(* CODESYS project Projekt_Wytwornia_Soku_Jerzy_Batygolski.project

Project tree, tasks and I/O mapping:
  Device : Berghof MX6 Control, Berghof Automation GmbH, version 1.21.0.0
    application Application
      libraries: Standard, 3.5.9.0 (System); Util, 3.5.11.0 (System); VisuUserMgmtDialogs, 3.5.10.0 (System); VisuDialogs, * (System); CAA Memory Block Manager Extern, 3.5.13.0 (CAA Technical Workgroup)
      task Control_program (cyclic, interval t#25ms, priority 1) calls CTRL_PRG
      task Simulation_program (cyclic, interval t#25ms, priority 1) calls SIM_PRG
      task VISU_TASK (cyclic, interval 50 ms, priority 31) calls VisuElems.Visu_Prg
      task TrendRecordingTask (cyclic, interval 100 ms, priority 31) calls VisuTrendStorageAccess.GlobalInstances.g_TrendRecordingManager.CyclicCall
      task AlarmManagerTask (cyclic, interval 50 ms, priority 31) calls AlarmManager.Alarm_Prg
      program SIM_PRG [ST]
      ENUMS/
        data type ConveyorStateEnum
        data type FillerStateEnum
        data type PasteurizationTankStateEnum
        data type PressStateEnum
        data type InnerFillerStateEnum
      MACHINE_STRUCTS/
        data type ConveyorMachineType
        data type PressMachineType
        data type PasteurizationTankType
        data type FillerMachineType
      STRUCTS/
        Conveyor/
          data type ConveyorCmdType
          data type ConveyorFailureType
          data type ConveyorSensorType
          data type ConveyorFlagType
          data type ConveyorParamType
        Press/
          data type PressCmdType
          data type PressFailureType
          data type PressSensorType
          data type PressFlagType
          data type PressParamType
        PasteurizationTank/
          data type PasteurCmdType
          data type PasteurFailureType
          data type PasteurSensorType
          data type PasteurFlagType
        Filler/
          data type FillerCmdType
          data type FillerFailureType
          data type FillerSensorType
          data type FillerFlagType
        Apple/
          data type AppleType
        Failure/
          data type FailureType
      image pool ImagePool
      program CTRL_PRG [ST]
      visualisation MainPage
      global variables GlobalVar
      visualisation Trends
      visualisation Alarms
      visualisation ErrorService
      Alarm Configuration
        alarm class ConvError (priority 10, acknowledge REP_ACK)
        alarm class TankLevelHigh (priority 30, acknowledge REP)
        AlarmStorage
        text list Conv
        alarm group Conv
            0 [ConvError]: Comparison Equal, ExpressionToCompare TRUE, Expression GlobalVar.Conveyor.Failure.ConvError.Active - "Conveyor is stuck"
            1 [GrinderError]: Comparison Equal, ExpressionToCompare TRUE, Expression GlobalVar.Conveyor.Failure.GrinderError.Active - "Grinder is stuck"
            2 [ConvEStop]: Comparison Equal, ExpressionToCompare TRUE, Expression GlobalVar.Conveyor.Failure.EStopPressed.Active - "Conveyor emergency stop is pressed"
            3 [GroundBuffer]: Comparison Equal, ExpressionToCompare TRUE, Expression GlobalVar.Conveyor.Failure.GroundBufferLevelTooHigh.Active - "Ground buffer level (<LATCH1> kg) is too high"
        alarm class GrinderError (priority 10, acknowledge REP_ACK)
        alarm class ConvEStop (priority 10, acknowledge REP_ACK)
        alarm class GroundBuffer (priority 10, acknowledge REP_ACK)
        alarm class PressError (priority 10, acknowledge REP_ACK)
        text list Press
        alarm group Press
            0 [PressError]: Comparison Equal, ExpressionToCompare TRUE, Expression GlobalVar.Press.Failure.PressError.Active - "Press is stucked"
            1 [TankBuffer]: Comparison Equal, ExpressionToCompare TRUE, Expression GlobalVar.Press.Failure.BufferTankLevelTooHigh.Active - "Buffer tank level (<LATCH1> l) is too high"
            2 [PressEStop]: Comparison Equal, ExpressionToCompare TRUE, Expression GlobalVar.Press.Failure.EStopPressed.Active - "Press emergency stop is pressed"
            3 [TankLevelHigh]: Comparison Equal, ExpressionToCompare TRUE, Expression GlobalVar.Press.Flag.TankLevelHigh - "Buffer tank level (<LATCH1> l) is high"
        text list PasteurizationTank
        alarm group PasteurizationTank
            0 [HeatingError]: Comparison Equal, ExpressionToCompare TRUE, Expression GlobalVar.PasteurTank.Failure.HeatingError.Active - "Heater is damaged"
            1 [PasteurEStop]: Comparison Equal, ExpressionToCompare TRUE, Expression GlobalVar.PasteurTank.Failure.EStopPressed.Active - "Pasteurization emergency stop is pressed"
        text list FillingMachine
        alarm group FillingMachine
            0 [CapError]: Comparison Equal, ExpressionToCompare TRUE, Expression GlobalVar.Filler.Failure.CapError.Active - "Cap is stuck"
            1 [FillError]: Comparison Equal, ExpressionToCompare TRUE, Expression GlobalVar.Filler.Failure.FillError.Active - "Filler is stuck"
            2 [FillerEStop]: Comparison Equal, ExpressionToCompare TRUE, Expression GlobalVar.Filler.Failure.EStopPressed.Active - "Filler emergency stop is pressed"
        alarm class TankBuffer (priority 10, acknowledge REP_ACK)
        alarm class PressEStop (priority 10, acknowledge REP_ACK)
        alarm class HeatingError (priority 10, acknowledge REP_ACK)
        alarm class PasteurEStop (priority 10, acknowledge REP_ACK)
        alarm class CapError (priority 10, acknowledge REP_ACK)
        alarm class FillError (priority 10, acknowledge REP_ACK)
        alarm class FillerEStop (priority 10, acknowledge REP_ACK)
  libraries: VisuSymbols, 3.5.10.0 (System)
  text list GlobalTextList
  5ce3da45-db07-42e7-a21c-a00fff4ed8f6|C:\Users\Jurek\Desktop\logo.png
  5ce3da45-db07-42e7-a21c-a00fff4ed8f6|C:\Users\Jurek\Desktop\Estop.png
  5ce3da45-db07-42e7-a21c-a00fff4ed8f6|C:\Users\Jurek\Desktop\Grafiki\EstopBtn2.jpg
  5ce3da45-db07-42e7-a21c-a00fff4ed8f6|C:\Users\Jurek\Desktop\Grafiki\EstopBtn2Pressed.jpg
  5ce3da45-db07-42e7-a21c-a00fff4ed8f6|C:\Users\Jurek\Desktop\Grafiki\Myjka_MT_1000.jpg
  5ce3da45-db07-42e7-a21c-a00fff4ed8f6|C:\Users\Jurek\Desktop\Grafiki\jablkaLevel3.png
  5ce3da45-db07-42e7-a21c-a00fff4ed8f6|C:\Users\Jurek\Desktop\Grafiki\jablkaLevel2.png
  5ce3da45-db07-42e7-a21c-a00fff4ed8f6|C:\Users\Jurek\Desktop\Grafiki\jablkaLevel1.png
  5ce3da45-db07-42e7-a21c-a00fff4ed8f6|C:\Users\Jurek\Desktop\Grafiki\jablkaLevel4.png
  5ce3da45-db07-42e7-a21c-a00fff4ed8f6|C:\Users\Jurek\Desktop\Grafiki\jablko5full.png
  5ce3da45-db07-42e7-a21c-a00fff4ed8f6|C:\Users\Jurek\Desktop\Grafiki\jablka_zmielone.png
  5ce3da45-db07-42e7-a21c-a00fff4ed8f6|C:\Users\Jurek\Desktop\Grafiki\prasaPNGgotowa.png
  5ce3da45-db07-42e7-a21c-a00fff4ed8f6|C:\Users\Jurek\Desktop\Grafiki\prasa\maleKolo.png
  5ce3da45-db07-42e7-a21c-a00fff4ed8f6|C:\Users\Jurek\Desktop\Grafiki\prasa\duzeKolo.png
  5ce3da45-db07-42e7-a21c-a00fff4ed8f6|C:\Users\Jurek\Desktop\Grafiki\prasa\nDuzeKolo.png
  5ce3da45-db07-42e7-a21c-a00fff4ed8f6|C:\Users\Jurek\Desktop\Grafiki\prasa\nMaleKolo.png
  5ce3da45-db07-42e7-a21c-a00fff4ed8f6|C:\Users\Jurek\Desktop\Grafiki\prasa\sok.png
  5ce3da45-db07-42e7-a21c-a00fff4ed8f6|C:\Users\Jurek\Desktop\Grafiki\prasa\zbiornik1500L.png
  5ce3da45-db07-42e7-a21c-a00fff4ed8f6|C:\Users\Jurek\Desktop\Grafiki\prasa\tank1000L.png
  5ce3da45-db07-42e7-a21c-a00fff4ed8f6|C:\Users\Jurek\Desktop\Grafiki\prasa\tank1002L.png
  5ce3da45-db07-42e7-a21c-a00fff4ed8f6|C:\Users\Jurek\Desktop\Grafiki\header.png
  5ce3da45-db07-42e7-a21c-a00fff4ed8f6|C:\Users\Jurek\Desktop\Grafiki\AlarmIcon.png
  5ce3da45-db07-42e7-a21c-a00fff4ed8f6|C:\Users\Jurek\Desktop\Grafiki\AlarmIcon2.png
*)

// Device/Application/ENUMS/ConveyorStateEnum
{attribute 'qualified_only'}
{attribute 'strict'}
TYPE ConveyorStateEnum :
(
	STATE_IDLE,
	STATE_WORKING,
	STATE_ERROR
);
END_TYPE

// Device/Application/ENUMS/FillerStateEnum
{attribute 'qualified_only'}
{attribute 'strict'}
TYPE FillerStateEnum :
(
	STATE_IDLE,
	STATE_WORKING,
	STATE_ERROR
);
END_TYPE

// Device/Application/ENUMS/PasteurizationTankStateEnum
{attribute 'qualified_only'}
{attribute 'strict'}
TYPE PasteurizationTankStateEnum :
(
	STATE_IDLE,
	STATE_FILLING,
	STATE_PASTEUR,
	STATE_ERROR
);
END_TYPE

// Device/Application/ENUMS/PressStateEnum
{attribute 'qualified_only'}
{attribute 'strict'}
TYPE PressStateEnum :
(
	STATE_IDLE,
	STATE_WORKING,
	STATE_ERROR
);
END_TYPE

// Device/Application/MACHINE_STRUCTS/ConveyorMachineType
TYPE ConveyorMachineType :
STRUCT
	Cmd: ConveyorCmdType;
	Failure: ConveyorFailureType;
	Sensor: ConveyorSensorType;
	State: ConveyorStateEnum;
	Flag: ConveyorFlagType;
	Param: ConveyorParamType;
END_STRUCT
END_TYPE

// Device/Application/MACHINE_STRUCTS/PressMachineType
TYPE PressMachineType :
STRUCT
	Cmd: PressCmdType;
	Failure: PressFailureType;
	Sensor: PressSensorType;
	State: PressStateEnum;
	Flag: PressFlagType;
	Param: PressParamType;
END_STRUCT
END_TYPE

// Device/Application/MACHINE_STRUCTS/PasteurizationTankType
TYPE PasteurizationTankType :
STRUCT
	Cmd: PasteurCmdType;
	Failure: PasteurFailureType;
	Sensor: PasteurSensorType;
	State: PasteurizationTankStateEnum;
	Flag: PasteurFlagType;
END_STRUCT
END_TYPE

// Device/Application/MACHINE_STRUCTS/FillerMachineType
TYPE FillerMachineType :
STRUCT
	Cmd: FillerCmdType;
	Failure: FillerFailureType;
	Sensor: FillerSensorType;
	State: FillerStateEnum;
	SimState: InnerFillerStateEnum;
	Flag: FillerFlagType;
END_STRUCT
END_TYPE

// Device/Application/STRUCTS/Conveyor/ConveyorCmdType
TYPE ConveyorCmdType :
STRUCT
	Start: BOOL;
	Stop: BOOL;
	EStop: BOOL;
	RunConv: BOOL;
END_STRUCT
END_TYPE

// Device/Application/STRUCTS/Conveyor/ConveyorFailureType
TYPE ConveyorFailureType :
STRUCT
	ConvError: FailureType;
	GrinderError: FailureType;
	EStopPressed: FailureType;
	GroundBufferLevelTooHigh: FailureType;
END_STRUCT
END_TYPE

// Device/Application/STRUCTS/Conveyor/ConveyorSensorType
TYPE ConveyorSensorType :
STRUCT
	Weight: REAL;
	GrinderRunning: BOOL;
END_STRUCT
END_TYPE

// Device/Application/STRUCTS/Conveyor/ConveyorFlagType
TYPE ConveyorFlagType :
STRUCT
	ProcessError: BOOL;
	ApplesOnConveyor: BOOL;
END_STRUCT
END_TYPE

// Device/Application/STRUCTS/Press/PressCmdType
TYPE PressCmdType :
STRUCT
	Start: BOOL;
	Stop: BOOL;
	EStop: BOOL;
	PressRun: BOOL;
END_STRUCT
END_TYPE

// Device/Application/STRUCTS/Press/PressFailureType
TYPE PressFailureType :
STRUCT
	PressError: FailureType;
	BufferTankLevelTooHigh: FailureType;
	EStopPressed: FailureType;
END_STRUCT
END_TYPE

// Device/Application/STRUCTS/Press/PressSensorType
TYPE PressSensorType :
STRUCT
	GroundBufferLevel: REAL;
	TotalJuiceProduced: REAL;
	TankLevel: REAL;
END_STRUCT
END_TYPE

// Device/Application/STRUCTS/Press/PressFlagType
TYPE PressFlagType :
STRUCT
	ProcessError: BOOL;
	TankLevelHigh: BOOL;
END_STRUCT
END_TYPE

// Device/Application/STRUCTS/PasteurizationTank/PasteurCmdType
TYPE PasteurCmdType :
STRUCT
	Start: BOOL;
	Stop: BOOL;
	EStop: BOOL;
	Fill: BOOL;
	Heat: BOOL;
	Cool: BOOL;
END_STRUCT
END_TYPE

// Device/Application/STRUCTS/PasteurizationTank/PasteurFailureType
TYPE PasteurFailureType :
STRUCT
	HeatingError: FailureType;
	EStopPressed: FailureType;
END_STRUCT
END_TYPE

// Device/Application/STRUCTS/PasteurizationTank/PasteurSensorType
TYPE PasteurSensorType :
STRUCT
	TankLevel: REAL;
	TargetTemp: REAL;
	ActTemp: LREAL;
END_STRUCT
END_TYPE

// Device/Application/STRUCTS/PasteurizationTank/PasteurFlagType
TYPE PasteurFlagType :
STRUCT
	ProcessError: BOOL;
	Filling: BOOL;
	Heating: BOOL;
	Cooling: BOOL;
END_STRUCT
END_TYPE

// Device/Application/STRUCTS/Filler/FillerCmdType
TYPE FillerCmdType :
STRUCT
	Start: BOOL;
	Stop: BOOL;
	EStop: BOOL;
	Run: BOOL;
END_STRUCT
END_TYPE

// Device/Application/STRUCTS/Filler/FillerFailureType
TYPE FillerFailureType :
STRUCT
	CapError: FailureType;
	FillError: FailureType;
	EStopPressed: FailureType;
END_STRUCT
END_TYPE

// Device/Application/STRUCTS/Filler/FillerSensorType
TYPE FillerSensorType :
STRUCT
	TankLevel: REAL;
	TotalProducedBottles: INT;
END_STRUCT
END_TYPE

// Device/Application/STRUCTS/Filler/FillerFlagType
TYPE FillerFlagType :
STRUCT
	ProcessError: BOOL;
	NewBottle: BOOL;
END_STRUCT
END_TYPE

// Device/Application/STRUCTS/Apple/AppleType
TYPE AppleType :
STRUCT
	Timer: TON;
	DX: INT;
	DY: INT;
	Invisible: BOOL;
END_STRUCT
END_TYPE

// Device/Application/STRUCTS/Conveyor/ConveyorParamType
TYPE ConveyorParamType :
STRUCT
	Speed: INT;
	GrindingRate: REAL;
END_STRUCT
END_TYPE

// Device/Application/STRUCTS/Press/PressParamType
TYPE PressParamType :
STRUCT
	JuiceProductionRate: REAL;
END_STRUCT
END_TYPE

// Device/Application/ENUMS/InnerFillerStateEnum
{attribute 'qualified_only'}
{attribute 'strict'}
TYPE InnerFillerStateEnum :
(
	STATE_RUN1,
	STATE_FILLING,
	STATE_CAPPING,
	STATE_RUN2,
	STATE_WAITING
);
END_TYPE

// Device/Application/STRUCTS/Failure/FailureType
TYPE FailureType :
STRUCT
	Active: BOOL;
	NeedAck: BOOL;
END_STRUCT
END_TYPE

// Device/Application/GlobalVar
{attribute 'qualified_only'}
VAR_GLOBAL
	Conveyor: ConveyorMachineType := (Param := (Speed := 1));
	Press: PressMachineType;
	PasteurTank: PasteurizationTankType := (Sensor := (TargetTemp := 78, ActTemp := 22));
	Filler: FillerMachineType;
	ActiveScreen: INT := 0;
END_VAR

// Device/Application/CTRL_PRG
PROGRAM CTRL_PRG
VAR
	YellowWarningInvisible: BOOL := TRUE;
	RedWarningInvisible: BOOL := TRUE;
END_VAR

(*
	Apple juice factory - control program
	Author: Jerzy Batygolski
	Date: 30.08.2018 
*)

(******************************************************************* Updating parameters ************************************************************************)

GlobalVar.Conveyor.Param.GrindingRate := GlobalVar.Conveyor.Param.Speed;
GlobalVar.Conveyor.Param.GrindingRate := GlobalVar.Conveyor.Param.GrindingRate / 100;
GlobalVar.Press.Param.JuiceProductionRate := GlobalVar.Conveyor.Param.GrindingRate / 1.5;

(*************************************************************** Checking if any errors has occured *************************************************************)

// Conveyor errors
GlobalVar.Conveyor.Failure.EStopPressed.Active := GlobalVar.Conveyor.Cmd.EStop;

IF GlobalVar.Press.Sensor.GroundBufferLevel >= 30 THEN
	GlobalVar.Conveyor.Failure.GroundBufferLevelTooHigh.Active := TRUE;
ELSE
	GlobalVar.Conveyor.Failure.GroundBufferLevelTooHigh.Active := FALSE;
END_IF;

IF (GlobalVar.Conveyor.Failure.ConvError.NeedAck OR GlobalVar.Conveyor.Failure.EStopPressed.NeedAck OR GlobalVar.Conveyor.Failure.GrinderError.NeedAck OR GlobalVar.Conveyor.Failure.GroundBufferLevelTooHigh.NeedAck) THEN
	GlobalVar.Conveyor.Flag.ProcessError := TRUE;
ELSE 
	GlobalVar.Conveyor.Flag.ProcessError := FALSE;
END_IF;

// Press errors
GlobalVar.Press.Failure.EStopPressed.Active := GlobalVar.Press.Cmd.EStop;

IF GlobalVar.Press.Sensor.TankLevel >= 97 THEN
	GlobalVar.Press.Failure.BufferTankLevelTooHigh.Active := TRUE;
ELSE 
	GlobalVar.Press.Failure.BufferTankLevelTooHigh.Active := FALSE;
END_IF;

IF GlobalVar.Press.Sensor.TankLevel >= 80 THEN
	GlobalVar.Press.Flag.TankLevelHigh := TRUE;
ELSE
	GlobalVar.Press.Flag.TankLevelHigh := FALSE;
END_IF;

IF (GlobalVar.Press.Failure.PressError.NeedAck OR GlobalVar.Press.Failure.BufferTankLevelTooHigh.NeedAck OR GlobalVar.Press.Failure.EStopPressed.NeedAck) THEN
	GlobalVar.Press.Flag.ProcessError := TRUE;
ELSE 
	GlobalVar.Press.Flag.ProcessError := FALSE;
END_IF;

// Pasteurization Tank errors
GlobalVar.PasteurTank.Failure.EStopPressed.Active := GlobalVar.PasteurTank.Cmd.EStop;
IF (GlobalVar.PasteurTank.Failure.EStopPressed.NeedAck OR GlobalVar.PasteurTank.Failure.HeatingError.NeedAck) THEN
	GlobalVar.PasteurTank.Flag.ProcessError := TRUE;
ELSE 
	GlobalVar.PasteurTank.Flag.ProcessError := FALSE;
END_IF;

// Filler machine errors
GlobalVar.Filler.Failure.EStopPressed.Active := GlobalVar.Filler.Cmd.EStop;
IF (GlobalVar.Filler.Failure.CapError.NeedAck OR GlobalVar.Filler.Failure.EStopPressed.NeedAck OR GlobalVar.Filler.Failure.FillError.NeedAck) THEN
	GlobalVar.Filler.Flag.ProcessError := TRUE;
ELSE
	GlobalVar.Filler.Flag.ProcessError := FALSE;
END_IF

// Updating warning icons visibility
IF (GlobalVar.Conveyor.Flag.ProcessError OR GlobalVar.Press.Flag.ProcessError OR GlobalVar.PasteurTank.Flag.ProcessError OR GlobalVar.Filler.Flag.ProcessError OR GlobalVar.Press.Flag.TankLevelHigh) THEN
	YellowWarningInvisible := FALSE;
ELSE
	YellowWarningInvisible := TRUE;
END_IF;

IF (GlobalVar.Conveyor.Failure.ConvError.Active OR GlobalVar.Conveyor.Failure.EStopPressed.Active OR GlobalVar.Conveyor.Failure.GrinderError.Active OR 
GlobalVar.Conveyor.Failure.GroundBufferLevelTooHigh.Active OR GlobalVar.Press.Failure.PressError.Active OR GlobalVar.Press.Failure.BufferTankLevelTooHigh.Active OR
GlobalVar.Press.Failure.EStopPressed.Active OR GlobalVar.PasteurTank.Failure.EStopPressed.Active OR GlobalVar.PasteurTank.Failure.HeatingError.Active OR
GlobalVar.Filler.Failure.CapError.Active OR GlobalVar.Filler.Failure.EStopPressed.Active OR GlobalVar.Filler.Failure.FillError.Active) THEN
	RedWarningInvisible := FALSE;
ELSE
	RedWarningInvisible := TRUE;
END_IF;

(*************************************************************** Conveyor state machine service *****************************************************************)

CASE GlobalVar.Conveyor.State OF
	
	ConveyorStateEnum.STATE_IDLE:
	
	IF GlobalVar.Conveyor.Flag.ProcessError THEN
		GlobalVar.Conveyor.State := ConveyorStateEnum.STATE_ERROR;
	ELSIF (GlobalVar.Conveyor.Sensor.Weight > 0 OR GlobalVar.Conveyor.Flag.ApplesOnConveyor) AND GlobalVar.Conveyor.Cmd.Start THEN
		GlobalVar.Conveyor.Cmd.RunConv := TRUE;
		GlobalVar.Conveyor.State := ConveyorStateEnum.STATE_WORKING;
	ELSIF GlobalVar.Conveyor.Cmd.Stop THEN
		GlobalVar.Conveyor.Cmd.Start := FALSE;
	END_IF;
	
	ConveyorStateEnum.STATE_WORKING:
	
	IF GlobalVar.Conveyor.Flag.ProcessError THEN
		GlobalVar.Conveyor.Cmd.RunConv := FALSE;
		GlobalVar.Conveyor.Cmd.Start := FALSE;
		GlobalVar.Conveyor.State := ConveyorStateEnum.STATE_ERROR;
	ELSIF GlobalVar.Conveyor.Cmd.Stop THEN
		GlobalVar.Conveyor.Cmd.Start := FALSE;
		GlobalVar.Conveyor.Cmd.RunConv := FALSE;
		GlobalVar.Conveyor.State := ConveyorStateEnum.STATE_IDLE;
	ELSIF GlobalVar.Conveyor.Sensor.Weight = 0 AND GlobalVar.Conveyor.Flag.ApplesOnConveyor = FALSE THEN
		GlobalVar.Conveyor.Cmd.RunConv := FALSE;
		GlobalVar.Conveyor.State := ConveyorStateEnum.STATE_IDLE;
	END_IF;
	
	ConveyorStateEnum.STATE_ERROR:
	
	GlobalVar.Conveyor.Cmd.Start := FALSE;
	GlobalVar.Conveyor.Cmd.Stop := FALSE;
	IF GlobalVar.Conveyor.Flag.ProcessError = FALSE THEN
		GlobalVar.Conveyor.State := ConveyorStateEnum.STATE_IDLE;
	END_IF;
	
END_CASE;

(*********************************************************** Press state machine service *********************************************************************)

CASE GlobalVar.Press.State OF
	
	PressStateEnum.STATE_IDLE:
	
	IF GlobalVar.Press.Flag.ProcessError THEN
		GlobalVar.Press.State := PressStateEnum.STATE_ERROR;
	ELSIF GlobalVar.Press.Cmd.Start AND GlobalVar.Press.Sensor.GroundBufferLevel > 0 THEN
		GlobalVar.Press.Cmd.PressRun := TRUE;
		GlobalVar.Press.State := PressStateEnum.STATE_WORKING;
	ELSIF GlobalVar.Press.Cmd.Stop THEN
		GlobalVar.Press.Cmd.Start := FALSE;
	END_IF;
	
	PressStateEnum.STATE_WORKING:
	
	IF GlobalVar.Press.Flag.ProcessError THEN
		GlobalVar.Press.Cmd.PressRun := FALSE;
		GlobalVar.Press.State := PressStateEnum.STATE_ERROR;
	ELSIF GlobalVar.Press.Cmd.Stop THEN
		GlobalVar.Press.Cmd.Start := FALSE;
		GlobalVar.Press.Cmd.PressRun := FALSE;
		GlobalVar.Press.State := PressStateEnum.STATE_IDLE;
	ELSIF GlobalVar.Press.Sensor.GroundBufferLevel = 0 THEN
		GlobalVar.Press.Cmd.PressRun := FALSE;
		GlobalVar.Press.State := PressStateEnum.STATE_IDLE;
	END_IF;
	
	PressStateEnum.STATE_ERROR:
	
	GlobalVar.Press.Cmd.Start := FALSE;
	GlobalVar.Press.Cmd.Stop := FALSE;
	IF GlobalVar.Press.Flag.ProcessError = FALSE THEN
		GlobalVar.Press.State := PressStateEnum.STATE_IDLE;
	END_IF;
	
END_CASE;

(*************************************************************** Pasteurization Tank state machine service *****************************************************)

CASE GlobalVar.PasteurTank.State OF
	
	PasteurizationTankStateEnum.STATE_IDLE:
	
	IF GlobalVar.PasteurTank.Flag.ProcessError THEN
		GlobalVar.PasteurTank.State := PasteurizationTankStateEnum.STATE_ERROR;
	ELSIF GlobalVar.PasteurTank.Cmd.Start AND GlobalVar.PasteurTank.Flag.Heating = FALSE AND GlobalVar.Press.Sensor.TankLevel > 0 THEN
		GlobalVar.PasteurTank.Flag.Filling := TRUE;
		GlobalVar.PasteurTank.Cmd.Fill := TRUE;
		GlobalVar.PasteurTank.State := PasteurizationTankStateEnum.STATE_FILLING;
	ELSIF GlobalVar.PasteurTank.Cmd.Start AND GlobalVar.PasteurTank.Flag.Heating THEN
		GlobalVar.PasteurTank.Cmd.Heat := TRUE;
		GlobalVar.PasteurTank.State := PasteurizationTankStateEnum.STATE_PASTEUR;
	ELSIF GlobalVar.PasteurTank.Cmd.Stop THEN
		GlobalVar.PasteurTank.Cmd.Start := FALSE;
	END_IF;
	
	PasteurizationTankStateEnum.STATE_FILLING:
	
	IF GlobalVar.PasteurTank.Flag.ProcessError THEN
		GlobalVar.PasteurTank.Cmd.Fill := FALSE;
		GlobalVar.PasteurTank.Cmd.Start := FALSE;
		GlobalVar.PasteurTank.State := PasteurizationTankStateEnum.STATE_ERROR;
	ELSIF GlobalVar.PasteurTank.Cmd.Stop THEN
		GlobalVar.PasteurTank.Cmd.Start := FALSE;
		GlobalVar.PasteurTank.Cmd.Fill := FALSE;
		GlobalVar.PasteurTank.State := PasteurizationTankStateEnum.STATE_IDLE;
	ELSIF (GlobalVar.PasteurTank.Sensor.TankLevel >= 10 AND GlobalVar.Press.Sensor.TankLevel = 0 AND GlobalVar.Press.Cmd.PressRun = FALSE) OR GlobalVar.PasteurTank.Sensor.TankLevel = 50 THEN
		GlobalVar.PasteurTank.Cmd.Fill := FALSE;
		GlobalVar.PasteurTank.Flag.Filling := FALSE;
		GlobalVar.PasteurTank.Cmd.Heat := TRUE;
		GlobalVar.PasteurTank.Flag.Heating := TRUE;
		GlobalVar.PasteurTank.State := PasteurizationTankStateEnum.STATE_PASTEUR;
	ELSIF GlobalVar.Press.Sensor.TankLevel = 0 THEN
		GlobalVar.PasteurTank.Cmd.Fill := FALSE;
		GlobalVar.PasteurTank.State := PasteurizationTankStateEnum.STATE_IDLE;
	END_IF;
	
	PasteurizationTankStateEnum.STATE_PASTEUR:
	
	IF GlobalVar.PasteurTank.Flag.ProcessError THEN
		GlobalVar.PasteurTank.Cmd.Heat := FALSE;
		GlobalVar.PasteurTank.Cmd.Start := FALSE;
		GlobalVar.PasteurTank.State := PasteurizationTankStateEnum.STATE_ERROR;
	ELSIF GlobalVar.PasteurTank.Cmd.Stop THEN
		GlobalVar.PasteurTank.Cmd.Start := FALSE;
		GlobalVar.PasteurTank.Cmd.Heat := FALSE;
		GlobalVar.PasteurTank.State := PasteurizationTankStateEnum.STATE_IDLE;
	ELSIF GlobalVar.PasteurTank.Sensor.TankLevel = 0 THEN
		GlobalVar.PasteurTank.Cmd.Heat := FALSE;
		GlobalVar.PasteurTank.Flag.Heating := FALSE;
		GlobalVar.PasteurTank.State := PasteurizationTankStateEnum.STATE_IDLE;
	END_IF;
	
	PasteurizationTankStateEnum.STATE_ERROR:
	
	GlobalVar.PasteurTank.Cmd.Start := FALSE;
	GlobalVar.PasteurTank.Cmd.Stop := FALSE;
	IF GlobalVar.PasteurTank.Flag.ProcessError = FALSE THEN
		GlobalVar.PasteurTank.State := PasteurizationTankStateEnum.STATE_IDLE;
	END_IF;
	
END_CASE;

(************************************************************** Filler state machine service *******************************************************************)

CASE GlobalVar.Filler.State OF
	
	FillerStateEnum.STATE_IDLE:
	
	IF GlobalVar.Filler.Flag.ProcessError THEN
		GlobalVar.Filler.State := FillerStateEnum.STATE_ERROR;
	ELSIF GlobalVar.Filler.Cmd.Start AND GlobalVar.Filler.Sensor.TankLevel >= 0.5 THEN
		GlobalVar.Filler.Cmd.Run := TRUE;
		GlobalVar.Filler.State := FillerStateEnum.STATE_WORKING;
	ELSIF GlobalVar.Filler.Cmd.Stop THEN
		GlobalVar.Filler.Cmd.Start := FALSE;
	END_IF;
	
	FillerStateEnum.STATE_WORKING:
	
	IF GlobalVar.Filler.Flag.ProcessError THEN
		GlobalVar.Filler.Cmd.Run := FALSE;
		GlobalVar.Filler.State := FillerStateEnum.STATE_ERROR;
	ELSIF GlobalVar.Filler.Cmd.Stop THEN
		GlobalVar.Filler.Cmd.Start := FALSE;
		GlobalVar.Filler.Cmd.Run := FALSE;
		GlobalVar.Filler.State := FillerStateEnum.STATE_IDLE;
	ELSIF GlobalVar.Filler.Sensor.TankLevel < 0.5 AND GlobalVar.Filler.Flag.NewBottle THEN
		GlobalVar.Filler.Cmd.Run := FALSE;
		GlobalVar.Filler.State := FillerStateEnum.STATE_IDLE;
	END_IF;
	
	FillerStateEnum.STATE_ERROR:
	
	GlobalVar.Filler.Cmd.Start := FALSE;
	GlobalVar.Filler.Cmd.Stop := FALSE;
	IF GlobalVar.Filler.Flag.ProcessError = FALSE THEN
		GlobalVar.Filler.State := FillerStateEnum.STATE_IDLE;
	END_IF;
	
END_CASE;

END_PROGRAM

// Device/Application/SIM_PRG
PROGRAM SIM_PRG
VAR
	PressEstopImg: STRING;
	FillerEstopImg: STRING;
	PasteurEstopImg: STRING;
	ConvEstopImg: STRING;
	ApplesImg: STRING;
	TimeConvCounter: INT := 1;
	GroundApples: AppleType := (Timer := (PT := TIME#800MS), Invisible := TRUE);
	ConvStopping: F_TRIG := (CLK := GlobalVar.Conveyor.Cmd.RunConv);
	ConvStarting: R_TRIG := (CLK := GlobalVar.Conveyor.Cmd.RunConv);
	TimerApples: TON := (PT := TIME#50ms);
	TimerEndConv: TON;
	Apples: ARRAY[0..3] OF AppleType := [4((Invisible := TRUE))];
	i: INT;
	BigRollerAngle: INT;
	SmallRollerAngle: INT;
	TimerPipes: TON := (PT := TIME#100ms);
	TimePipesCounter: INT;
	Pipes1Invisible: ARRAY[0..6] OF BOOL := [7(TRUE)];
	EndJuice: F_TRIG;
	StartJuice: R_TRIG;
	EndJuiceMarker: BOOL;
	TimeJuiceProduction: INT;
	Pipes2Invisible: BOOL := TRUE;
	PasteurStartFill: R_TRIG;
	PasteurEndFill: F_TRIG;
	Tout: REAL := 295;
	T0: LREAL := 295;
	A: REAL := 70;
	B: REAL := 8;
	HeatStop: F_TRIG;
	HeatStart: R_TRIG;
	TimerHeating: TON := (IN := TRUE, PT := TIME#100ms);
	TimeHeatingCounter: REAL := 0.0;
	Pipes3Invisible: BOOL := TRUE;
	HeatingLamp: BOOL := FALSE;
	BottleInvisible: BOOL := FALSE;
	CapInvisible: BOOL := TRUE;
	JuiceInvisible: ARRAY[0..2] OF BOOL := [3(TRUE)];
	FillerInvisible: BOOL := TRUE;
	BottleDX: INT;
	CapDY: INT;
	TimeFilling: INT;
	TraceBufferTankLevel: BOOL := FALSE;
	TracePasteurTemp: BOOL := FALSE;
	TraceProducedBottles: BOOL := FALSE;
	Timer: TON := (IN := TRUE, PT := TIME#1s0ms);
	SecondsElapsed: INT;
	MinutesElapsed: INT;
	ProductionRate: INT;
END_VAR

(*
	Apple juice factory - simulation program
	Author: Jerzy Batygolski
	Date: 30.08.2018 
*)

(*************************************************************** Updating parameters *****************************************************************)

TimerEndConv.PT := TIME#450MS / GlobalVar.Conveyor.Param.Speed;
Timer.IN := TRUE;
Timer();
IF Timer.Q THEN
	Timer.IN := FALSE;
	Timer();
	SecondsElapsed := SecondsElapsed + 1;
	IF SecondsElapsed = 60 THEN
		MinutesElapsed := MinutesElapsed + 1;
		SecondsElapsed := 0;
	END_IF;
END_IF;

IF MinutesElapsed > 0 THEN
	ProductionRate := GlobalVar.Filler.Sensor.TotalProducedBottles / MinutesElapsed;
ELSE
	ProductionRate := 0;
END_IF;

(********************************************************* EStop button simulation *******************************************************************)

IF GlobalVar.Conveyor.Cmd.EStop THEN
	ConvEstopImg := 'ImagePool.EStopPressed';
ELSE
	ConvEstopImg := 'ImagePool.EStop';
END_IF;

IF GlobalVar.Press.Cmd.EStop THEN
	PressEstopImg := 'ImagePool.EStopPressed';
ELSE
	PressEstopImg := 'ImagePool.EStop';
END_IF;

IF GlobalVar.PasteurTank.Cmd.EStop THEN
	PasteurEstopImg := 'ImagePool.EStopPressed';
ELSE
	PasteurEstopImg := 'ImagePool.EStop';
END_IF;

IF GlobalVar.Filler.Cmd.EStop THEN
	FillerEstopImg := 'ImagePool.EStopPressed';
ELSE
	FillerEstopImg := 'ImagePool.EStop';
END_IF;

(********************************************************* Conveyor simulation ***************************************************************)

// Apples container simulation
IF GlobalVar.Conveyor.Sensor.Weight = 0 THEN
	ApplesImg := '';
ELSIF GlobalVar.Conveyor.Sensor.Weight > 0 AND GlobalVar.Conveyor.Sensor.Weight <= 5 THEN
	ApplesImg := 'ImagePool.jablkaLevel1';
ELSIF GlobalVar.Conveyor.Sensor.Weight > 5 AND GlobalVar.Conveyor.Sensor.Weight <= 10 THEN
	ApplesImg := 'ImagePool.jablkaLevel2';
ELSIF GlobalVar.Conveyor.Sensor.Weight > 10 AND GlobalVar.Conveyor.Sensor.Weight <= 20 THEN
	ApplesImg := 'ImagePool.jablkaLevel3';
ELSIF GlobalVar.Conveyor.Sensor.Weight > 20 THEN
	ApplesImg := 'ImagePool.jablkaLevel4';
END_IF;

// Apples on conveyor simulation
// Conveyor starting
ConvStarting.CLK := GlobalVar.Conveyor.Cmd.RunConv;
ConvStarting();
IF ConvStarting.Q THEN
	GlobalVar.Conveyor.Flag.ApplesOnConveyor := TRUE;
	IF GlobalVar.Conveyor.Sensor.Weight > 0 THEN
		Apples[0].Invisible := FALSE;
	END_IF;
END_IF;

// Conveyor stopping
ConvStopping.CLK := GlobalVar.Conveyor.Cmd.RunConv;
ConvStopping();
IF ConvStopping.Q THEN
	GroundApples.Invisible := TRUE;
	GlobalVar.Conveyor.Sensor.GrinderRunning := FALSE;
END_IF;

// Conveyor running
IF GlobalVar.Conveyor.Cmd.RunConv THEN
	
	IF TimerEndConv.IN = FALSE AND GlobalVar.Conveyor.Flag.ApplesOnConveyor THEN
		
		TimerApples.IN := TRUE;
		TimerApples();
		IF TimerApples.Q THEN
			TimerApples.IN := FALSE;
			TimerApples();
			TimeConvCounter := TimeConvCounter + 1 * GlobalVar.Conveyor.Param.Speed;
			FOR	i := 0 TO 3 DO
				IF TimeConvCounter > (i * 15) THEN
				
					IF GlobalVar.Conveyor.Sensor.Weight > 0 THEN
						Apples[i].Invisible := FALSE;
					END_IF;
				
					IF Apples[i].Invisible = FALSE THEN
						Apples[i].DX := Apples[i].DX + 3 * GlobalVar.Conveyor.Param.Speed;
						Apples[i].DY := Apples[i].DY - 4 * GlobalVar.Conveyor.Param.Speed;
					END_IF;
				
					IF Apples[i].DX > 177 THEN
						IF GlobalVar.Conveyor.Sensor.Weight = 0 THEN
							Apples[i].Invisible := TRUE;
							IF Apples[0].Invisible AND Apples[1].Invisible AND Apples[2].Invisible AND Apples[3].Invisible THEN
								TimerApples.IN := FALSE;
								TimerApples(); 
								TimerEndConv.IN := TRUE;
								TimerEndConv();
							END_IF;
						END_IF;
						Apples[i].DX := 0;
						Apples[i].DY := 0;
					END_IF;
				
				END_IF;
			END_FOR;
		
			IF TimeConvCounter > 66  THEN
				GlobalVar.Conveyor.Sensor.GrinderRunning := TRUE;
			END_IF;
		END_IF;
	
		GlobalVar.Conveyor.Sensor.Weight := GlobalVar.Conveyor.Sensor.Weight - GlobalVar.Conveyor.Param.GrindingRate;
		IF GlobalVar.Conveyor.Sensor.Weight < 0 THEN
			GlobalVar.Conveyor.Sensor.Weight := 0;
		END_IF;
		
	END_IF;
	
	TimerEndConv();
	IF TimerEndConv.Q THEN
		TimerEndConv.IN := FALSE;
		TimerEndConv();
		GlobalVar.Conveyor.Flag.ApplesOnConveyor := FALSE;
		TimeConvCounter := 1;
	END_IF;
	
END_IF;

// Grinder simulation
IF GlobalVar.Conveyor.Sensor.GrinderRunning THEN
	GroundApples.Timer.IN := TRUE;
	GroundApples.Timer();
	IF GroundApples.Timer.Q THEN
		GroundApples.Invisible := NOT(GroundApples.Invisible);
		GroundApples.Timer.IN := FALSE;
		GroundApples.Timer();
	END_IF;
	GlobalVar.Press.Sensor.GroundBufferLevel := GlobalVar.Press.Sensor.GroundBufferLevel + GlobalVar.Conveyor.Param.GrindingRate;
END_IF;

(******************************************************** Press simulation ****************************************************************)

IF GlobalVar.Press.Cmd.PressRun THEN
	
	// Rollers simulaton
	BigRollerAngle := BigRollerAngle + 1;
	SmallRollerAngle := SmallRollerAngle - 1;
	IF BigRollerAngle = 360 THEN
		BigRollerAngle := 0;
	END_IF;
	IF SmallRollerAngle = -360 THEN
		SmallRollerAngle := 0;
	END_IF;
	
	// Ground buffer simulation
	GlobalVar.Press.Sensor.GroundBufferLevel := GlobalVar.Press.Sensor.GroundBufferLevel - GlobalVar.Conveyor.Param.GrindingRate;
	IF GlobalVar.Press.Sensor.GroundBufferLevel < 0 THEN
		GlobalVar.Press.Sensor.GroundBufferLevel := 0;
	END_IF;
	
	GlobalVar.Press.Sensor.TotalJuiceProduced := GlobalVar.Press.Sensor.TotalJuiceProduced + GlobalVar.Press.Param.JuiceProductionRate;
	
	// Pipes and buffer simulation
	TimerPipes.IN := TRUE;
	TimerPipes();
	IF TimerPipes.Q THEN
		TimerPipes.IN := FALSE;
		TimerPipes();
		TimePipesCounter := TimePipesCounter + 1;
		TimeJuiceProduction := TimeJuiceProduction + 1;
		IF TimePipesCounter = 5 THEN
			Pipes1Invisible[0] := FALSE;
			Pipes1Invisible[1] := FALSE;
		ELSIF TimePipesCounter = 12 THEN
			Pipes1Invisible[2] := FALSE;
			Pipes1Invisible[3] := FALSE;
		ELSIF TimePipesCounter = 19 THEN
			Pipes1Invisible[4] := FALSE;
			Pipes1Invisible[5] := FALSE;
		ELSIF TimePipesCounter = 26 THEN
			Pipes1Invisible[6] := FALSE;
		END_IF;
	END_IF;
	
	IF TimePipesCounter > 26 THEN
		GlobalVar.Press.Sensor.TankLevel := GlobalVar.Press.Sensor.TankLevel + GlobalVar.Press.Param.JuiceProductionRate;
	ELSE 
		GlobalVar.Press.Cmd.Stop := FALSE;
	END_IF;
	
END_IF;

// Start juice production
StartJuice.CLK := GlobalVar.Press.Cmd.PressRun;
StartJuice();
IF StartJuice.Q THEN
	TimeJuiceProduction := 0;
END_IF;

// End juice production
EndJuice.CLK := GlobalVar.Press.Cmd.PressRun;
EndJuice();
IF EndJuice.Q THEN
	TimePipesCounter := 0;
	EndJuiceMarker := TRUE;
	IF TimeJuiceProduction > 26 THEN
		TimeJuiceProduction := 26;
	END_IF;
END_IF;

IF EndJuiceMarker THEN
	TimerPipes.IN := TRUE;
	TimerPipes();
	IF TimerPipes.Q THEN
		TimerPipes.IN := FALSE;
		TimerPipes();
		TimePipesCounter := TimePipesCounter + 1;
		IF TimePipesCounter = 5 THEN
			Pipes1Invisible[0] := TRUE;
			Pipes1Invisible[1] := TRUE;
		ELSIF TimePipesCounter = 12 THEN
			Pipes1Invisible[2] := TRUE;
			Pipes1Invisible[3] := TRUE;
		ELSIF TimePipesCounter = 19 THEN
			Pipes1Invisible[4] := TRUE;
			Pipes1Invisible[5] := TRUE;
		ELSIF TimePipesCounter = 26 THEN
			Pipes1Invisible[6] := TRUE;
		END_IF;
	END_IF;
	
	IF TimePipesCounter <= TimeJuiceProduction THEN
		GlobalVar.Press.Sensor.TankLevel := GlobalVar.Press.Sensor.TankLevel + GlobalVar.Press.Param.JuiceProductionRate;
	ELSE 
		EndJuiceMarker := FALSE;
		TimerPipes.IN := FALSE;
		TimerPipes();
		TimePipesCounter := 0;
	END_IF;
	
END_IF;

(******************************************************* Pasteurization process simulation **********************************************************)

// Filling simulation
PasteurStartFill.CLK := GlobalVar.PasteurTank.Cmd.Fill;
PasteurStartFill();
IF PasteurStartFill.Q THEN
	Pipes2Invisible := FALSE;
END_IF;

PasteurEndFill.CLK := GlobalVar.PasteurTank.Cmd.Fill;
PasteurEndFill();
IF PasteurEndFill.Q THEN
	Pipes2Invisible := TRUE;
END_IF;

IF GlobalVar.PasteurTank.Cmd.Fill THEN
	GlobalVar.PasteurTank.Sensor.TankLevel := GlobalVar.PasteurTank.Sensor.TankLevel + GlobalVar.Press.Param.JuiceProductionRate;
	IF GlobalVar.PasteurTank.Sensor.TankLevel > 50 THEN
		GlobalVar.PasteurTank.Sensor.TankLevel := 50;
	END_IF;
	GlobalVar.Press.Sensor.TankLevel := GlobalVar.Press.Sensor.TankLevel - GlobalVar.Press.Param.JuiceProductionRate;
	IF GlobalVar.Press.Sensor.TankLevel < 0 THEN
		GlobalVar.Press.Sensor.TankLevel := 0;
	END_IF;
END_IF;

// Heating simulation
IF GlobalVar.PasteurTank.Cmd.Heat AND GlobalVar.PasteurTank.Flag.Cooling = FALSE THEN
	HeatingLamp := TRUE;
ELSE HeatingLamp := FALSE;
END_IF;

HeatStart.CLK := GlobalVar.PasteurTank.Cmd.Heat;
HeatStart();
IF HeatStart.Q THEN
	T0 := GlobalVar.PasteurTank.Sensor.ActTemp + 273;
	TimeHeatingCounter := 0;
END_IF;

HeatStop.CLK := GlobalVar.PasteurTank.Cmd.Heat;
HeatStop();
IF HeatStop.Q THEN
	TimeHeatingCounter := 0;
	T0 := GlobalVar.PasteurTank.Sensor.ActTemp + 273;
END_IF;

TimerHeating.IN := TRUE;
TimerHeating();

IF TimerHeating.Q THEN
	TimerHeating.IN := FALSE;
	TimerHeating();
	TimeHeatingCounter := TimeHeatingCounter + 0.01 * GlobalVar.Conveyor.Param.Speed;
	IF GlobalVar.PasteurTank.Flag.Cooling = FALSE AND GlobalVar.PasteurTank.Cmd.Heat THEN
		// heating
		GlobalVar.PasteurTank.Sensor.ActTemp := Tout + A - 273 - ((Tout - T0 + A) / EXPT(2.718, B / GlobalVar.PasteurTank.Sensor.TankLevel * TimeHeatingCounter));
		IF GlobalVar.PasteurTank.Sensor.ActTemp >= GlobalVar.PasteurTank.Sensor.TargetTemp THEN
			GlobalVar.PasteurTank.Sensor.ActTemp := GlobalVar.PasteurTank.Sensor.TargetTemp;
			GlobalVar.PasteurTank.Flag.Cooling := TRUE;
			TimeHeatingCounter := 0;
			T0 := GlobalVar.PasteurTank.Sensor.ActTemp + 273;
		END_IF;
	ELSIF GlobalVar.PasteurTank.Flag.Cooling = TRUE AND GlobalVar.PasteurTank.Cmd.Heat THEN
		// pasteurization
		IF GlobalVar.PasteurTank.Sensor.ActTemp < GlobalVar.PasteurTank.Sensor.TargetTemp AND TimeHeatingCounter <= 0.24 THEN
			TimeHeatingCounter := 0.25;
		END_IF;
		IF TimeHeatingCounter > 0.24 THEN
			// cooling
			GlobalVar.PasteurTank.Sensor.ActTemp := Tout  - 273 - ((Tout - T0) / EXPT(2.718, B / GlobalVar.PasteurTank.Sensor.TankLevel * (TimeHeatingCounter - 0.24)));
		END_IF;
	ELSIF GlobalVar.PasteurTank.Cmd.Heat = FALSE THEN
		GlobalVar.PasteurTank.Sensor.ActTemp := Tout  - 273 - ((Tout - T0) / EXPT(2.718, B / GlobalVar.PasteurTank.Sensor.TankLevel * TimeHeatingCounter));
	END_IF;
END_IF;
IF GlobalVar.PasteurTank.Flag.Cooling AND GlobalVar.PasteurTank.Cmd.Heat AND (GlobalVar.PasteurTank.Sensor.ActTemp + 273) <= (Tout + 6) AND GlobalVar.PasteurTank.Sensor.TankLevel > 0 THEN
	GlobalVar.PasteurTank.Sensor.TankLevel := GlobalVar.PasteurTank.Sensor.TankLevel - GlobalVar.Press.Param.JuiceProductionRate;
	Pipes3Invisible := FALSE;
	GlobalVar.Filler.Sensor.TankLevel := GlobalVar.Filler.Sensor.TankLevel + GlobalVar.Press.Param.JuiceProductionRate;
	IF GlobalVar.PasteurTank.Sensor.TankLevel <= 0 THEN
		GlobalVar.PasteurTank.Sensor.TankLevel := 0;
		GlobalVar.PasteurTank.Flag.Cooling := FALSE;
		Pipes3Invisible := TRUE;
		TimeHeatingCounter := 0;
	END_IF;
END_IF;

(****************************************************** Filling process simulation *************************************************************)
IF GlobalVar.Filler.Cmd.Run THEN
	CASE GlobalVar.Filler.SimState OF
		
	InnerFillerStateEnum.STATE_RUN1:
	
	BottleDX := BottleDX + 1 * GlobalVar.Conveyor.Param.Speed;
	IF BottleDx >= 69 THEN
		FillerInvisible := FALSE;
		GlobalVar.Filler.Flag.NewBottle := FALSE;
		GlobalVar.Filler.SimState := InnerFillerStateEnum.STATE_FILLING;
	END_IF;
	
	InnerFillerStateEnum.STATE_FILLING:
	
	TimeFilling := TimeFilling + 1 * GlobalVar.Conveyor.Param.Speed;
	IF TimeFilling >= 80 THEN
		FillerInvisible := TRUE;
		JuiceInvisible[1] := TRUE;
		JuiceInvisible[2] := FALSE;
		CapInvisible := FALSE;
		GlobalVar.Filler.Sensor.TankLevel := globalvar.Filler.Sensor.TankLevel - 0.5;
		GlobalVar.Filler.SimState := InnerFillerStateEnum.STATE_CAPPING;
	ELSIF TimeFilling >= 50 THEN
		JuiceInvisible[0] := TRUE;
		JuiceInvisible[1] := FALSE;
	ELSIF TimeFilling >= 20 THEN
		JuiceInvisible[0] := FALSE;
	END_IF;
	
	InnerFillerStateEnum.STATE_CAPPING:
	
	CapDY := CapDY + 1 * GlobalVar.Conveyor.Param.Speed;
	IF CapDy >= 30 THEN
		TimeFilling := 0;
		GlobalVar.Filler.SimState := InnerFillerStateEnum.STATE_RUN2;
	END_IF;
	
	InnerFillerStateEnum.STATE_RUN2:
	
	BottleDX := BottleDX + 1 * GlobalVar.Conveyor.Param.Speed;
	IF BottleDX >= 140 THEN
		BottleInvisible := TRUE;
		JuiceInvisible[2] := TRUE;
		CapInvisible := TRUE;
		BottleDX := 0;
		CapDY := 0;
		TimeFilling := 0;
		GlobalVar.Filler.Sensor.TotalProducedBottles := GlobalVar.Filler.Sensor.TotalProducedBottles + 1;
		GlobalVar.Filler.SimState := InnerFillerStateEnum.STATE_WAITING;
	END_IF;
		
	InnerFillerStateEnum.STATE_WAITING:
	TimeFilling := TimeFilling + 1 * GlobalVar.Conveyor.Param.Speed;
	IF TimeFilling >= 20 THEN
		TimeFilling := 0;
		BottleInvisible := FALSE;
		GlobalVar.Filler.Flag.NewBottle := TRUE;
		GlobalVar.Filler.SimState := InnerFillerStateEnum.STATE_RUN1;
	END_IF;
	
	END_CASE;
END_IF;

END_PROGRAM

// Device/Application/MainPage
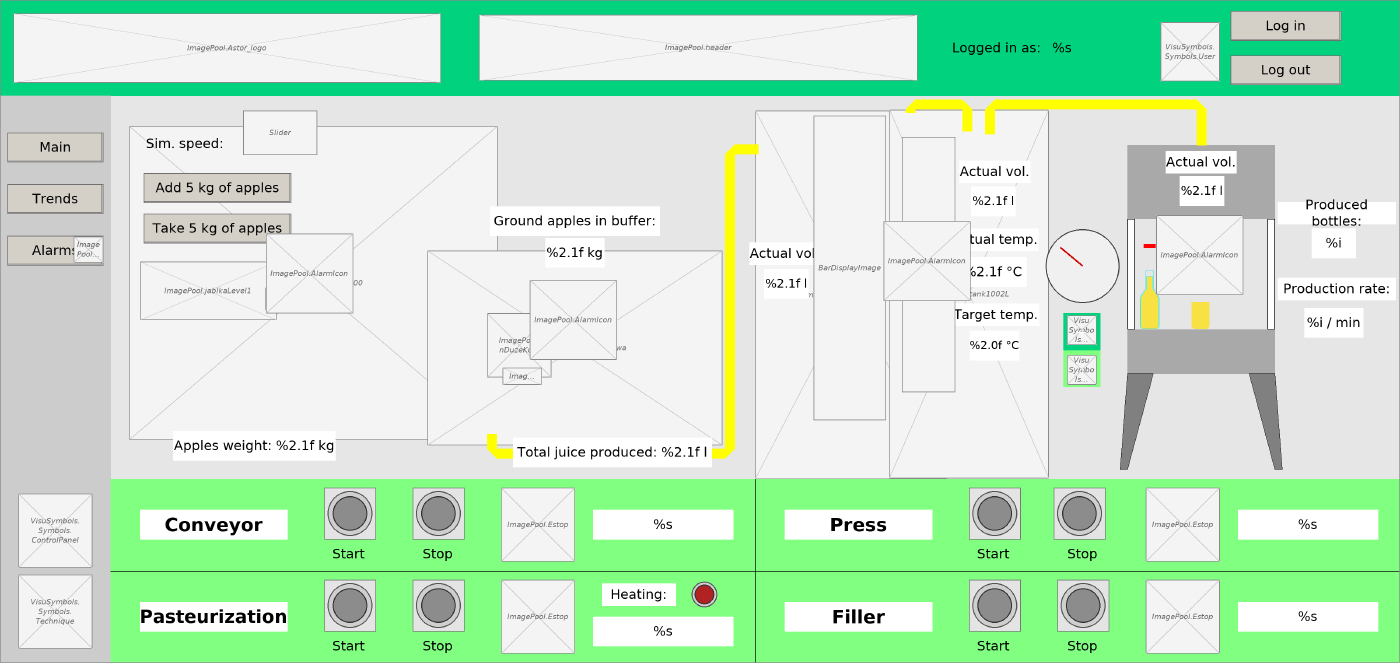
VISUALIZATION MainPage  // 1900x900
    Image (1025,150 260x500), image: ImagePool.zbiornik1500L
    Image (1207,149 216x500), image: ImagePool.tank1002L
    Polygon (1617,443) (1620,446) (1638,446) (1641,443) (1641,410) (1617,410), invisible if: SIM_PRG.JuiceInvisible[1]
    Polygon (1617,443) (1620,446) (1638,446) (1641,443) (1641,433) (1617,433), invisible if: SIM_PRG.JuiceInvisible[0]
    Polygon (1548,405) (1550,400) (1555,393) (1556,391) (1556,375) (1564,375) (1564,391) (1565,393) (1570,400) (1572,405) (1572,443) (1569,446) (1551,446) (1548,443), invisible if: SIM_PRG.JuiceInvisible[2]
        p3560616238: SIM_PRG.BottleDX
    Polygon (1547,404) (1549,399) (1554,392) (1555,389) (1555,367) (1565,367) (1565,389) (1566,392) (1571,399) (1573,404) (1573,444) (1570,447) (1550,447) (1547,444), invisible if: SIM_PRG.BottleInvisible
        p3560616238: SIM_PRG.BottleDX
    Polygon (1306,148) (1306,135) (1319,148)
    Polygon (1229,148) (1242,135) (1242,148)
    Polygon (1229,148) (1242,135) (1242,148), invisible if: SIM_PRG.Pipes2Invisible
    Polygon (1306,148) (1306,135) (1319,148), invisible if: SIM_PRG.Pipes2Invisible
    Rectangle (1443,475 50x50)
    Image (190,395 189x29), image: ImagePool.jablkaLevel1
    Rectangle (0,0 1900x130)
    Rectangle (0,130 150x770)
    Image (18,18 580x94), image: ImagePool.Astor_logo
    Rectangle (150,650 1750x250)
    Label (423,737 100x30), "Start"
    Line (150,775) (1900,775)
    Line (1025,650) (1025,900)
    Image (680,662 100x100), image: ImagePool.Estop
        p84334746: SIM_PRG.ConvEstopImg
        OnMouseDown:  ToggleVariable=GlobalVar.Conveyor.Cmd.EStop
    Rectangle (190,692 200x40), "Conveyor"
    Label (544,737 100x30), "Stop"
    Image (175,171 500x426), image: ImagePool.Myjka_MT_1000
    Rectangle (805,692 190x40), "%s", text variable: GlobalVar.Conveyor.State
    Rectangle (235,585 220x40), "Apples weight: %2.1f kg", text variable: GlobalVar.Conveyor.Sensor.Weight
    Button (195,235 200x40), "Add 5 kg of apples"
        OnMouseClick: execute { GlobalVar.Conveyor.Sensor.Weight := GlobalVar.Conveyor.Sensor.Weight + 5; }
    Button (195,290 200x40), "Take 5 kg of apples"
        OnMouseClick: execute {
            IF GlobalVar.Conveyor.Sensor.Weight >= 5 THEN
            GlobalVar.Conveyor.Sensor.Weight := GlobalVar.Conveyor.Sensor.Weight - 5;
            END_IF;
        }
    Image (190,355 185x79), image: ImagePool.jablkaLevel1
        p84334746: SIM_PRG.ApplesImg
    Slider (330,150 100x60), variable: GlobalVar.Conveyor.Param.Speed, scale 1..3
    Label (195,180 130x30), "Sim. speed:"
    Image (360,390 29x31), invisible if: SIM_PRG.Apples[0].Invisible, image: ImagePool.jablko
        p3560616238: SIM_PRG.Apples[0].DX
        p2738717112: SIM_PRG.Apples[0].DY
    Image (360,390 29x31), invisible if: SIM_PRG.Apples[1].Invisible, image: ImagePool.jablko
        p3560616238: SIM_PRG.Apples[1].DX
        p2738717112: SIM_PRG.Apples[1].DY
    Image (360,390 29x31), invisible if: SIM_PRG.Apples[2].Invisible, image: ImagePool.jablko
        p3560616238: SIM_PRG.Apples[2].DX
        p2738717112: SIM_PRG.Apples[2].DY
    Image (360,390 29x31), invisible if: SIM_PRG.Apples[3].Invisible, image: ImagePool.jablko
        p3560616238: SIM_PRG.Apples[3].DX
        p2738717112: SIM_PRG.Apples[3].DY
    PushSwitch (440,662 70x70), variable: GlobalVar.Conveyor.Cmd.Start, behaviour: TOGGLE, style: Switch-PushSwitch-Gray
    PushSwitch (560,662 70x70), variable: GlobalVar.Conveyor.Cmd.Stop, behaviour: TAP, style: Switch-PushSwitch-Gray
    Image (610,350 45x25), invisible if: SIM_PRG.GroundApples.Invisible, image: ImagePool.jablka_zmielone
        p3560616238: SIM_PRG.GroundApples.DX
        p2738717112: SIM_PRG.GroundApples.DY
    Rectangle (1065,692 200x40), "Press"
    PushSwitch (1315,662 70x70), variable: GlobalVar.Press.Cmd.Start, behaviour: TOGGLE, style: Switch-PushSwitch-Gray
    PushSwitch (1430,662 70x70), variable: GlobalVar.Press.Cmd.Stop, behaviour: TAP, style: Switch-PushSwitch-Gray
    Label (1298,737 100x30), "Start"
    Label (1419,737 100x30), "Stop"
    Image (1555,662 100x100), image: ImagePool.Estop
        p84334746: SIM_PRG.PressEstopImg
        OnMouseDown:  ToggleVariable=GlobalVar.Press.Cmd.EStop
    Rectangle (1680,692 190x40), "%s", text variable: GlobalVar.Press.State
    Rectangle (190,817 200x40), "Pasteurization"
    Rectangle (1065,817 200x40), "Filler"
    PushSwitch (440,787 70x70), variable: GlobalVar.PasteurTank.Cmd.Start, behaviour: TOGGLE, style: Switch-PushSwitch-Gray
    PushSwitch (560,787 70x70), variable: GlobalVar.PasteurTank.Cmd.Stop, behaviour: TAP, style: Switch-PushSwitch-Gray
    Image (680,787 100x100), image: ImagePool.Estop
        p84334746: SIM_PRG.PasteurEstopImg
        OnMouseDown:  ToggleVariable=GlobalVar.PasteurTank.Cmd.EStop
    Rectangle (805,837 190x40), "%s", text variable: GlobalVar.PasteurTank.State
    Label (423,862 100x30), "Start"
    Label (544,862 100x30), "Stop"
    PushSwitch (1315,787 70x70), variable: GlobalVar.Filler.Cmd.Start, behaviour: TOGGLE, style: Switch-PushSwitch-Gray
    PushSwitch (1435,787 70x70), variable: GlobalVar.Filler.Cmd.Stop, behaviour: TAP, style: Switch-PushSwitch-Gray
    Image (1555,787 100x100), image: ImagePool.Estop
        p84334746: SIM_PRG.FillerEstopImg
        OnMouseDown:  ToggleVariable=GlobalVar.Filler.Cmd.EStop
    Rectangle (1680,817 190x40), "%s", text variable: GlobalVar.Filler.State
    Label (1298,862 100x30), "Start"
    Label (1419,862 100x30), "Stop"
    Image (580,340 400x264), image: ImagePool.prasaPNGgotowa
    Image (661,425 87x87), image: ImagePool.nDuzeKolo
        p2858320360: SIM_PRG.BigRollerAngle
    Image (737,413 47x47), image: ImagePool.nMaleKolo
        p2858320360: SIM_PRG.SmallRollerAngle
    Image (682,499 53x23), invisible if: NOT(GlobalVar.Press.Cmd.PressRun), image: ImagePool.sok
    Rectangle (674,609 310x13)
    Rectangle (661,589 13x20)
    Polygon (661,609) (674,609) (674,622)
    Polygon (984,609) (997,609) (984,622)
    Rectangle (984,209 13x400)
    Polygon (984,209) (997,196) (997,209)
    Rectangle (997,196 32x13)
    Rectangle (1229,148 13x5)
    Rectangle (1242,135 64x13)
    Rectangle (1306,148 13x30)
    Rectangle (665,280 230x40), "Ground apples in buffer:"
    Rectangle (740,323 80x40), "%2.1f kg", text variable: GlobalVar.Press.Sensor.GroundBufferLevel
    Rectangle (661,589 13x20), invisible if: SIM_PRG.Pipes1Invisible[0]
    Polygon (661,609) (674,609) (674,622), invisible if: SIM_PRG.Pipes1Invisible[1]
    Rectangle (674,609 310x13), invisible if: SIM_PRG.Pipes1Invisible[2]
    Rectangle (696,594 270x40), "Total juice produced: %2.1f l", text variable: GlobalVar.Press.Sensor.TotalJuiceProduced, invisible if: TRUE
    Polygon (984,609) (997,609) (984,622), invisible if: SIM_PRG.Pipes1Invisible[3]
    Rectangle (984,209 13x400), invisible if: SIM_PRG.Pipes1Invisible[4]
    Polygon (984,209) (997,196) (997,209), invisible if: SIM_PRG.Pipes1Invisible[5]
    Rectangle (997,196 32x13), invisible if: SIM_PRG.Pipes1Invisible[6]
    Rectangle (1037,365 60x40), "%2.1f l", text variable: GlobalVar.Press.Sensor.TankLevel
    Rectangle (1302,349 91x40), "%2.1f °C", text variable: GlobalVar.PasteurTank.Sensor.ActTemp
    Rectangle (1316,449 67x40), "%2.0f °C", text variable: GlobalVar.PasteurTank.Sensor.TargetTemp
    Rectangle (1302,218 96x30), "Actual vol."
    Rectangle (1318,253 60x40), "%2.1f l", text variable: GlobalVar.PasteurTank.Sensor.TankLevel
    Rectangle (1443,425 50x50)
    Image (1448,428 40x40), image: VisuSymbols.Symbols.TriangleUp
        OnMouseClick: execute { GlobalVar.PasteurTank.Sensor.TargetTemp := GlobalVar.PasteurTank.Sensor.TargetTemp + 1; }
    Image (1448,482 40x40), image: VisuSymbols.Symbols.TriangleDown
        OnMouseClick: execute { GlobalVar.PasteurTank.Sensor.TargetTemp := GlobalVar.PasteurTank.Sensor.TargetTemp - 1; }
    Label (1456,436 25x30), "+"
    Label (1456,485 25x30), "-"
    Rectangle (1229,148 13x5), invisible if: SIM_PRG.Pipes2Invisible
    Rectangle (1242,135 64x13), invisible if: SIM_PRG.Pipes2Invisible
    Rectangle (1306,148 13x30), invisible if: SIM_PRG.Pipes2Invisible
    Rectangle (1530,297 10x150)
    Rectangle (1720,297 10x150)
    Rectangle (1530,447 200x60)
    Rectangle (1530,197 200x100)
    Polygon (1530,507) (1565,507) (1530,637) (1520,637)
    Polygon (1695,507) (1730,507) (1740,637) (1730,637)
    Rectangle (1337,148 13x34)
    Polygon (1337,148) (1350,135) (1350,148)
    Rectangle (1350,135 274x13)
    Rectangle (1624,148 13x49)
    Polygon (1624,148) (1624,135) (1637,148)
    Rectangle (1582,205 96x30), "Actual vol."
    Rectangle (1601,239 60x40), "%2.1f l", text variable: GlobalVar.Filler.Sensor.TankLevel
    Rectangle (1337,148 13x34), invisible if: SIM_PRG.Pipes3Invisible
    Rectangle (1350,135 274x13), invisible if: SIM_PRG.Pipes3Invisible
    Rectangle (1624,148 13x49), invisible if: SIM_PRG.Pipes3Invisible
    Polygon (1337,148) (1350,135) (1350,148), invisible if: SIM_PRG.Pipes3Invisible
    Polygon (1624,148) (1624,135) (1637,148), invisible if: SIM_PRG.Pipes3Invisible
    Rectangle (1734,274 160x30), "Produced bottles:"
    Rectangle (1780,310 60x40), "%i", text variable: GlobalVar.Filler.Sensor.TotalProducedBottles
    Polygon (1623,297) (1634,297) (1634,350) (1629,360) (1623,350)
    Polygon (1623,297) (1634,297) (1634,350) (1629,360) (1623,350), invisible if: SIM_PRG.FillerInvisible
    Rectangle (1552,331 16x5), invisible if: SIM_PRG.CapInvisible
        p2738717112: SIM_PRG.CapDY
        p3560616238: SIM_PRG.BottleDX
    Rectangle (1017,329 96x30), "Actual vol."
    Meter360 (1419,311 100x100), value: GlobalVar.PasteurTank.Sensor.ActTemp, style: Meter-Meter360-Green, scale format: %.0f, scale 20..100
        p518627256: °C
    Rectangle (817,792 100x30), "Heating:"
    Lamp1 (936,787 40x40), variable: SIM_PRG.HeatingLamp, style: Lamp-Lamp1-Red
    Rectangle (1292,310 117x30), "Actual temp."
    Rectangle (1293,412 117x30), "Target temp."
    BarDisplayImage (1224,186 72x346), value: GlobalVar.PasteurTank.Sensor.TankLevel, style: BarDisplayImage-Blue, scale format: %.1f, scale 0..50
        p518627256: Litres
    BarDisplayImage (1104,157 98x413), value: GlobalVar.Press.Sensor.TankLevel, style: BarDisplayImage-Yellow, scale format: %.1f, scale 0..100
        p518627256: Litres
    Image (650,20 595x89), image: ImagePool.header
    Button (10,250 130x40), "Trends", colour toggle: GlobalVar.ActiveScreen = 1
        OnMouseClick:  Assign=Trends, Type=Assignment
        OnMouseClick: execute { GlobalVar.ActiveScreen := 1; }
        OnMouseClick:  Dialog=ErrorService, Result=OK, NumpadKeypadSet=True
    Button (10,320 130x40), "Alarms", colour toggle: GlobalVar.ActiveScreen = 2
        OnMouseClick:  Assign=Alarms, Type=Assignment
        OnMouseClick: execute { GlobalVar.ActiveScreen := 2; }
        OnMouseClick:  Dialog=ErrorService, Result=OK, NumpadKeypadSet=True
    Button (1670,15 150x40), "Log in"
        OnMouseClick:  Type=Login
    Button (1670,75 150x40), "Log out"
        OnMouseClick:  Type=Logout
    Image (1575,30 80x80), image: VisuSymbols.Symbols.User
    Button (10,180 130x40), "Main", colour toggle: GlobalVar.ActiveScreen = 0
        OnMouseClick:  Assign=MainPage, Type=Assignment
        OnMouseClick: execute { GlobalVar.ActiveScreen := 0; }
    Rectangle (1289,50 275x30), "Logged in as:"
    Rectangle (1425,50 130x30), "%s", text variable: VisuNativeControl.CurrentFullUserName
    Image (25,780 100x100), image: VisuSymbols.Symbols.Technique
        OnMouseClick:  Dialog=ErrorService, PositionX=150, PositionY=650
    Image (25,670 100x100), image: VisuSymbols.Symbols.ControlPanel
        OnMouseClick:  Dialog=ErrorService, Result=OK, NumpadKeypadSet=True
    Image (361,317 118x108), invisible if: NOT(GlobalVar.Conveyor.Flag.ProcessError), image: ImagePool.AlarmIcon
    Image (719,380 118x108), invisible if: NOT(GlobalVar.Press.Flag.ProcessError), image: ImagePool.AlarmIcon
    Image (1199,300 118x108), invisible if: NOT(GlobalVar.PasteurTank.Flag.ProcessError), image: ImagePool.AlarmIcon
    Image (1569,292 118x108), invisible if: NOT(GlobalVar.Filler.Flag.ProcessError), image: ImagePool.AlarmIcon
    Image (100,321 40x35), invisible if: CTRL_PRG.YellowWarningInvisible, image: ImagePool.AlarmIcon2
    Image (100,321 40x35), invisible if: CTRL_PRG.RedWarningInvisible, image: ImagePool.AlarmIcon
    Rectangle (1734,377 160x30), "Production rate:"
    Rectangle (1770,418 80x40), "%i / min", text variable: SIM_PRG.ProductionRate
END_VISUALIZATION

// Device/Application/Trends
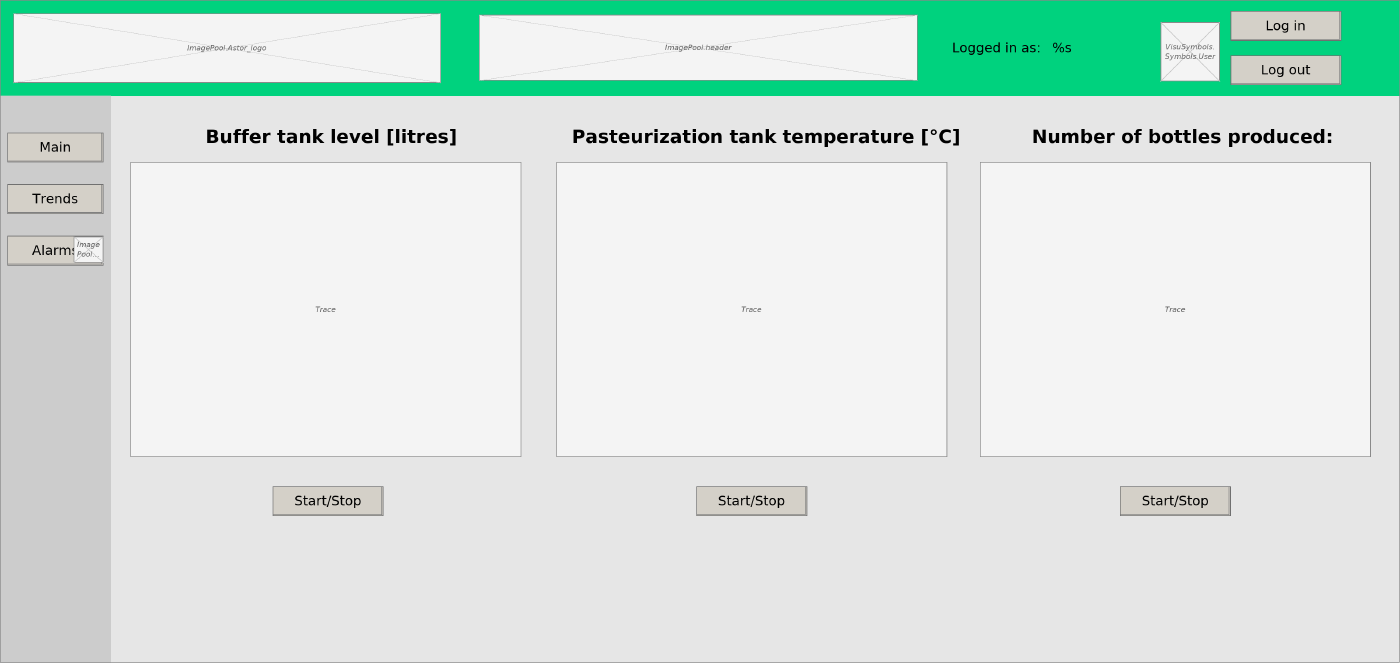
VISUALIZATION Trends  // 1900x900
    Rectangle (0,0 1900x130)
    Rectangle (0,130 150x770)
    Image (18,18 580x94), image: ImagePool.Astor_logo
    Image (650,20 595x89), image: ImagePool.header
    Button (10,250 130x40), "Trends", colour toggle: GlobalVar.ActiveScreen = 1
        OnMouseClick:  Assign=Trends, Type=Assignment
        OnMouseClick: execute { GlobalVar.ActiveScreen := 1; }
    Button (10,320 130x40), "Alarms", colour toggle: GlobalVar.ActiveScreen = 2
        OnMouseClick:  Assign=Alarms, Type=Assignment
        OnMouseClick: execute { GlobalVar.ActiveScreen := 2; }
    Button (10,180 130x40), "Main", colour toggle: GlobalVar.ActiveScreen = 0
        OnMouseClick:  Assign=MainPage, Type=Assignment
        OnMouseClick: execute { GlobalVar.ActiveScreen := 0; }
    Trace (177,220 530x400)
        p866368322: SIM_PRG.TraceBufferTankLevel = TRUE
        p3851742229: SIM_PRG.TraceBufferTankLevel = FALSE
    Button (370,660 150x40), "Start/Stop", colour toggle: SIM_PRG.TraceBufferTankLevel
        OnMouseClick:  ToggleVariable=SIM_PRG.TraceBufferTankLevel
    Label (275,170 350x30), "Buffer tank level [litres]"
    Trace (755,220 530x400)
        p866368322: SIM_PRG.TracePasteurTemp = TRUE
        p3851742229: SIM_PRG.TracePasteurTemp = FALSE
    Trace (1330,220 530x400)
        p866368322: SIM_PRG.TraceProducedBottles = TRUE
        p3851742229: SIM_PRG.TraceProducedBottles = FALSE
    Button (945,660 150x40), "Start/Stop", colour toggle: SIM_PRG.TracePasteurTemp
        OnMouseClick:  ToggleVariable=SIM_PRG.TracePasteurTemp
    Button (1520,660 150x40), "Start/Stop", colour toggle: SIM_PRG.TraceProducedBottles
        OnMouseClick:  ToggleVariable=SIM_PRG.TraceProducedBottles
    Label (790,170 500x30), "Pasteurization tank temperature [°C]"
    Label (1405,170 400x30), "Number of bottles produced:"
    Button (1670,15 150x40), "Log in"
        OnMouseClick:  Type=Login
    Button (1670,75 150x40), "Log out"
        OnMouseClick:  Type=Logout
    Image (1575,30 80x80), image: VisuSymbols.Symbols.User
    Rectangle (1289,50 275x30), "Logged in as:"
    Rectangle (1425,50 130x30), "%s", text variable: VisuNativeControl.CurrentFullUserName
    Image (100,321 40x35), invisible if: CTRL_PRG.YellowWarningInvisible, image: ImagePool.AlarmIcon2
    Image (100,321 40x35), invisible if: CTRL_PRG.RedWarningInvisible, image: ImagePool.AlarmIcon
END_VISUALIZATION

// Device/Application/Alarms
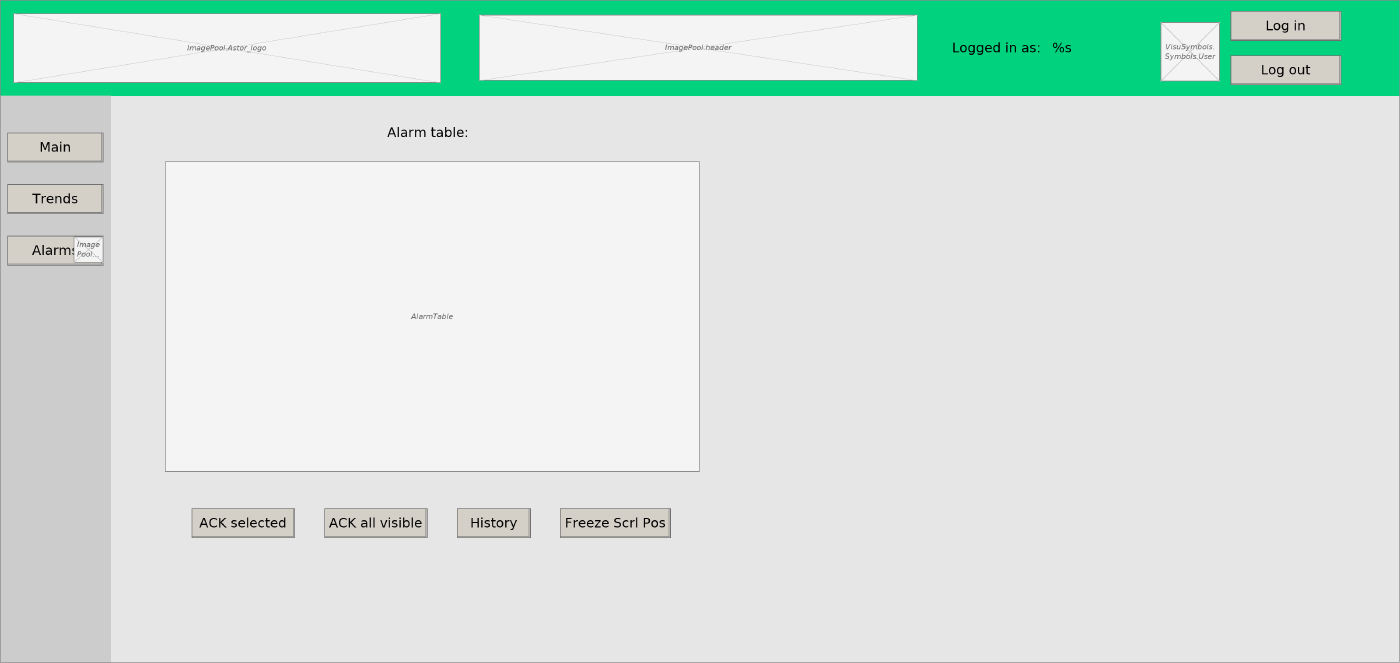
VISUALIZATION Alarms  // 1900x900
VAR_IN_OUT
END_VAR
VAR
	bAckSel : BOOL;
	bAckVisible : BOOL;
	bHistory : BOOL;
	bFreezeScrlPos : BOOL;
	bAckSel2 : BOOL;
END_VAR
    Rectangle (0,0 1900x130)
    Rectangle (0,130 150x770)
    Image (18,18 580x94), image: ImagePool.Astor_logo
    Image (650,20 595x89), image: ImagePool.header
    Button (10,250 130x40), "Trends", colour toggle: GlobalVar.ActiveScreen = 1
        OnMouseClick:  Assign=Trends, Type=Assignment
        OnMouseClick: execute { GlobalVar.ActiveScreen := 1; }
    Button (10,320 130x40), "Alarms", colour toggle: GlobalVar.ActiveScreen = 2
        OnMouseClick:  Assign=Alarms, Type=Assignment
        OnMouseClick: execute { GlobalVar.ActiveScreen := 2; }
    Button (10,180 130x40), "Main", colour toggle: GlobalVar.ActiveScreen = 0
        OnMouseClick:  Assign=MainPage, Type=Assignment
        OnMouseClick: execute { GlobalVar.ActiveScreen := 0; }
    Button (1670,15 150x40), "Log in"
        OnMouseClick:  Type=Login
    Button (1670,75 150x40), "Log out"
        OnMouseClick:  Type=Logout
    Image (1575,30 80x80), image: VisuSymbols.Symbols.User
    Rectangle (1289,50 275x30), "Logged in as:"
    Rectangle (1425,50 130x30), "%s", text variable: VisuNativeControl.CurrentFullUserName
    AlarmTable (224,219 725x421)
        Column[2]: ColumnTitle=Status
        Column[3]: ColumnTitle=Priority
        p1521930926: __All
        p1663851261: __All
        p428520879: bAckSel
        p2607059081: bAckVisible
        p3266827225: bHistory
        p3894972949: bFreezeScrlPos
    Label (481,165 200x30), "Alarm table:"
    Button (260,690 140x40), "ACK selected"
        toggle bAckSel
    Button (440,690 140x40), "ACK all visible"
        toggle bAckVisible
    Button (620,690 100x40), "History"
        toggle bHistory
    Button (760,690 150x40), "Freeze Scrl Pos"
        toggle bFreezeScrlPos
    Image (100,321 40x35), invisible if: CTRL_PRG.YellowWarningInvisible, image: ImagePool.AlarmIcon2
    Image (100,321 40x35), invisible if: CTRL_PRG.RedWarningInvisible, image: ImagePool.AlarmIcon
END_VISUALIZATION

// Device/Application/ErrorService
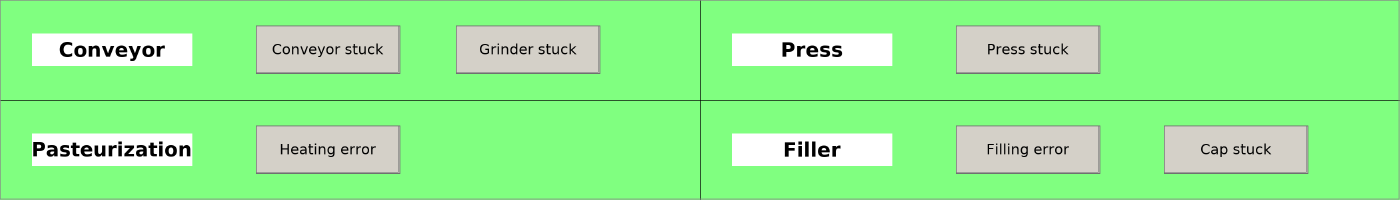
VISUALIZATION ErrorService  // 1750x250
    Rectangle (0,0 1750x250)
    Line (0,125) (1750,125)
    Line (875,0) (875,250)
    Rectangle (40,42 200x40), "Conveyor"
    Rectangle (40,167 200x40), "Pasteurization"
    Rectangle (915,42 200x40), "Press"
    Rectangle (915,167 200x40), "Filler"
    Button (320,32 180x60), "Conveyor stuck", colour toggle: GlobalVar.Conveyor.Failure.ConvError.Active
        OnMouseClick:  ToggleVariable=GlobalVar.Conveyor.Failure.ConvError.Active
    Button (570,32 180x60), "Grinder stuck", colour toggle: GlobalVar.Conveyor.Failure.GrinderError.Active
        OnMouseClick:  ToggleVariable=GlobalVar.Conveyor.Failure.GrinderError.Active
    Button (1195,32 180x60), "Press stuck", colour toggle: GlobalVar.Press.Failure.PressError.Active
        OnMouseClick:  ToggleVariable=GlobalVar.Press.Failure.PressError.Active
    Button (320,157 180x60), "Heating error", colour toggle: GlobalVar.PasteurTank.Failure.HeatingError.Active
        OnMouseClick:  ToggleVariable=GlobalVar.PasteurTank.Failure.HeatingError.Active
    Button (1195,157 180x60), "Filling error", colour toggle: GlobalVar.Filler.Failure.FillError.Active
        OnMouseClick:  ToggleVariable=GlobalVar.Filler.Failure.FillError.Active
    Button (1455,157 180x60), "Cap stuck", colour toggle: GlobalVar.Filler.Failure.CapError.Active
        OnMouseClick:  ToggleVariable=GlobalVar.Filler.Failure.CapError.Active
END_VISUALIZATION

(* text list Conv (id | default)
  3 | Ground buffer level (<LATCH1> kg) is too high
  2 | Conveyor emergency stop is pressed
  1 | Grinder is stuck
  0 | Conveyor is stuck
   |  *)

(* text list Press (id | default)
  3 | Buffer tank level (<LATCH1> l) is high
  2 | Press emergency stop is pressed
  1 | Buffer tank level (<LATCH1> l) is too high
  0 | Press is stucked
   |  *)

(* text list PasteurizationTank (id | default)
  1 | Pasteurization emergency stop is pressed
  0 | Heater is damaged
   |  *)

(* text list FillingMachine (id | default)
  2 | Filler emergency stop is pressed
  1 | Filler is stuck
  0 | Cap is stuck
   |  *)
